{attribute 'GeneratedUsingTerminal: EPP3174-0002-0016'}
{attribute addProperty BoxType "EPP3174-0002-0016"}
{attribute addProperty Id "AI_Standard_Channel_1AT %I*AI_Standard_Channel_A8DF64E310AI_Standard_Channel_2AT %I*AI_Standard_Channel_A8DF64E310AI_Standard_Channel_3AT %I*AI_Standard_Channel_A8DF64E310AI_Standard_Channel_4AT %I*AI_Standard_Channel_A8DF64E310WcStateAT %I*WcState_9091E0EB2InfoDataAT %I*InfoData_32EB74EA10"}
{attribute addProperty CRC "3704063586"}
{attribute addProperty Size "52"}
TYPE EPP3174_DCC78662 :
STRUCT
	{attribute addProperty Name "AI_Standard_Channel_1"}
	AI_Standard_Channel_1 : AI_Standard_Channel_A8DF64E3;
	{attribute addProperty Name "AI_Standard_Channel_2"}
	AI_Standard_Channel_2 : AI_Standard_Channel_A8DF64E3;
	{attribute addProperty Name "AI_Standard_Channel_3"}
	AI_Standard_Channel_3 : AI_Standard_Channel_A8DF64E3;
	{attribute addProperty Name "AI_Standard_Channel_4"}
	AI_Standard_Channel_4 : AI_Standard_Channel_A8DF64E3;
	{attribute addProperty Name "WcState"}
	WcState : WcState_9091E0EB;
	{attribute addProperty Name "InfoData"}
	InfoData : InfoData_32EB74EA;
END_STRUCT
END_TYPE

(* stored: Version 1.2.0.0, ProductVersion 3.1.4024.9
   DUT EPP3174_DCC78662: Id {50a1c65b-ae1c-4774-9d95-5fc33af2cbad} *)
